FUNCTION_BLOCK FireDamper EXTENDS Damper
VAR_INPUT
END_VAR
VAR_OUTPUT
END_VAR
VAR
END_VAR

END_FUNCTION_BLOCK

(* stored: Version 1.1.0.1, ProductVersion 3.1.4024.3
   POU FireDamper: Id {83eb272c-0be2-4677-9ef1-4597c43233af}, SpecialFunc None *)
